FUNCTION_BLOCK CNV_1_CONTROL (* Basic Function Block Type *)
  (* Standard: 61499-2 *)
  (* Version 0.3, 2009-09-15, JHC, Holobloc Inc, Changed transition priorities. *)
  (* Version 0.2, 2003-12-04, JHC, Rockwell Automation, Renamed for better indexing. *)
  (* Version 0.1, 2002-11-05, JHC, Rockwell Automation, Corrected missing ST element in Algorithm REQ. *)
  (* Version 0.0, 2000-05-30, JHC, Rockwell Automation *)
  (* Compiler header: package fb.rt.dasdA1.A2; *)
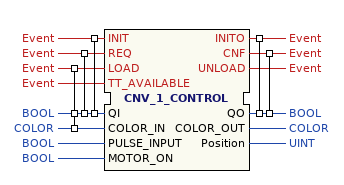
  EVENT_INPUT
    INIT WITH QI; (* Initialization Request *)
    REQ WITH QI; (* Normal Execution Request *)
    LOAD WITH COLOR_IN, QI;
    TT_AVAILABLE;
  END_EVENT
  EVENT_OUTPUT
    INITO WITH QO; (* Initialization Confirm *)
    CNF WITH QO; (* Execution Confirmation *)
    UNLOAD;
  END_EVENT
  VAR_INPUT
    QI : BOOL; (* Input event qualifier *)
    COLOR_IN : COLOR;
    PULSE_INPUT : BOOL;
    MOTOR_ON : BOOL;
  END_VAR
  VAR_OUTPUT
    QO : BOOL; (* Output event qualifier *)
    COLOR_OUT : COLOR;
    Position : UINT;
  END_VAR
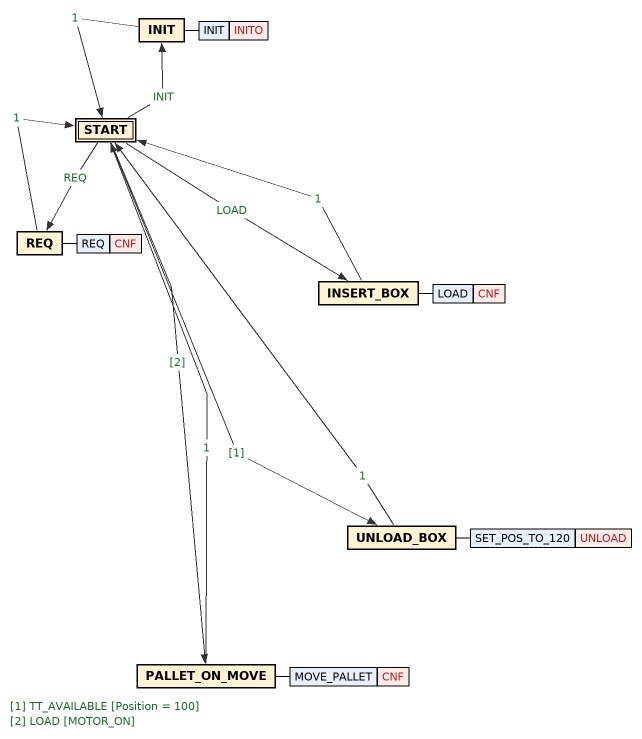
  EC_STATES
    START; (* Initial State *)
    INIT : INIT -> INITO; (* Initialization *)
    REQ : REQ -> CNF; (* Normal execution *)
    INSERT_BOX : LOAD -> CNF;
    UNLOAD_BOX : SET_POS_TO_120 -> UNLOAD;
    PALLET_ON_MOVE : MOVE_PALLET -> CNF;
  END_STATES
  EC_TRANSITIONS
    INIT TO START := 1;
    START TO REQ := REQ;
    START TO INIT := INIT;
    REQ TO START := 1;
    START TO INSERT_BOX := LOAD;
    INSERT_BOX TO START := 1;
    START TO UNLOAD_BOX := TT_AVAILABLE [Position = 100];
    UNLOAD_BOX TO START := 1;
    START TO PALLET_ON_MOVE := LOAD [MOTOR_ON];
    PALLET_ON_MOVE TO START := 1;
  END_TRANSITIONS
  ALGORITHM INIT IN ST: (* Initialization algorithm *)

  END_ALGORITHM
  ALGORITHM REQ IN ST: (* Normally executed algorithm *)

  END_ALGORITHM
  ALGORITHM LOAD IN ST:
COLOR_IN := COLOR_OUT;
  END_ALGORITHM
  ALGORITHM SET_POS_TO_120 IN ST:
IF Position = 100 THEN
Position := 120;
COLOR_OUT := null;
END_IF;
  END_ALGORITHM
  ALGORITHM MOVE_PALLET IN ST:
//INT COUNT = 0;
//WHILE Position <= 100; DO
//IF PULSE_INPUT THEN
//COUNT := COUNT + 1;
//Position := Position + COUNT*0.001;
//ELSE
//END_IF;
//END_WHILE;
  END_ALGORITHM
END_FUNCTION_BLOCK
